    "t" := ("x" - "g1_6"["lo"]) / ("g1_6"["hi"] - "g1_6"["lo"] + 1.0E-10);
    "class_1" := "class_1" + ("t1_1_6"["lo"] * (1.0 - "t") + "t1_1_6"["hi"] * "t");
    "class_2" := "class_2" + ("t1_2_6"["lo"] * (1.0 - "t") + "t1_2_6"["hi"] * "t");
    "class_3" := "class_3" + ("t1_3_6"["lo"] * (1.0 - "t") + "t1_3_6"["hi"] * "t");
    "class_4" := "class_4" + ("t1_4_6"["lo"] * (1.0 - "t") + "t1_4_6"["hi"] * "t");
    // input 7: binary search on L1 grid
    "lo" := 0; "hi" := 15;
    "x" := "h1_7";
    IF "x" < -3.15 THEN "x" := -3.15; END_IF;
    IF "x" > 3.15 THEN "x" := 3.15; END_IF;
    WHILE "hi" - "lo" > 1 DO
        "mid" := "lo" + ("hi" - "lo") / 2;
        IF "x" > "g1_7"["mid"] THEN "lo" := "mid"; ELSE "hi" := "mid"; END_IF;
    END_WHILE;
    "t" := ("x" - "g1_7"["lo"]) / ("g1_7"["hi"] - "g1_7"["lo"] + 1.0E-10);
    "class_1" := "class_1" + ("t1_1_7"["lo"] * (1.0 - "t") + "t1_1_7"["hi"] * "t");
    "class_2" := "class_2" + ("t1_2_7"["lo"] * (1.0 - "t") + "t1_2_7"["hi"] * "t");
    "class_3" := "class_3" + ("t1_3_7"["lo"] * (1.0 - "t") + "t1_3_7"["hi"] * "t");
    "class_4" := "class_4" + ("t1_4_7"["lo"] * (1.0 - "t") + "t1_4_7"["hi"] * "t");
    // input 8: binary search on L1 grid
    "lo" := 0; "hi" := 15;
    "x" := "h1_8";
    IF "x" < -3.15 THEN "x" := -3.15; END_IF;
    IF "x" > 3.15 THEN "x" := 3.15; END_IF;
    WHILE "hi" - "lo" > 1 DO
        "mid" := "lo" + ("hi" - "lo") / 2;
        IF "x" > "g1_8"["mid"] THEN "lo" := "mid"; ELSE "hi" := "mid"; END_IF;
    END_WHILE;
    "t" := ("x" - "g1_8"["lo"]) / ("g1_8"["hi"] - "g1_8"["lo"] + 1.0E-10);
    "class_1" := "class_1" + ("t1_1_8"["lo"] * (1.0 - "t") + "t1_1_8"["hi"] * "t");
    "class_2" := "class_2" + ("t1_2_8"["lo"] * (1.0 - "t") + "t1_2_8"["hi"] * "t");
    "class_3" := "class_3" + ("t1_3_8"["lo"] * (1.0 - "t") + "t1_3_8"["hi"] * "t");
    "class_4" := "class_4" + ("t1_4_8"["lo"] * (1.0 - "t") + "t1_4_8"["hi"] * "t");
    // input 9: binary search on L1 grid
    "lo" := 0; "hi" := 15;
    "x" := "h1_9";
    IF "x" < -3.15 THEN "x" := -3.15; END_IF;
    IF "x" > 3.15 THEN "x" := 3.15; END_IF;
    WHILE "hi" - "lo" > 1 DO
        "mid" := "lo" + ("hi" - "lo") / 2;
        IF "x" > "g1_9"["mid"] THEN "lo" := "mid"; ELSE "hi" := "mid"; END_IF;
    END_WHILE;
    "t" := ("x" - "g1_9"["lo"]) / ("g1_9"["hi"] - "g1_9"["lo"] + 1.0E-10);
    "class_1" := "class_1" + ("t1_1_9"["lo"] * (1.0 - "t") + "t1_1_9"["hi"] * "t");
    "class_2" := "class_2" + ("t1_2_9"["lo"] * (1.0 - "t") + "t1_2_9"["hi"] * "t");
    "class_3" := "class_3" + ("t1_3_9"["lo"] * (1.0 - "t") + "t1_3_9"["hi"] * "t");
    "class_4" := "class_4" + ("t1_4_9"["lo"] * (1.0 - "t") + "t1_4_9"["hi"] * "t");
    // input 10: binary search on L1 grid
    "lo" := 0; "hi" := 15;
    "x" := "h1_10";
    IF "x" < -3.15 THEN "x" := -3.15; END_IF;
    IF "x" > 3.15 THEN "x" := 3.15; END_IF;
    WHILE "hi" - "lo" > 1 DO
        "mid" := "lo" + ("hi" - "lo") / 2;
        IF "x" > "g1_10"["mid"] THEN "lo" := "mid"; ELSE "hi" := "mid"; END_IF;
    END_WHILE;
    "t" := ("x" - "g1_10"["lo"]) / ("g1_10"["hi"] - "g1_10"["lo"] + 1.0E-10);
    "class_1" := "class_1" + ("t1_1_10"["lo"] * (1.0 - "t") + "t1_1_10"["hi"] * "t");
    "class_2" := "class_2" + ("t1_2_10"["lo"] * (1.0 - "t") + "t1_2_10"["hi"] * "t");
    "class_3" := "class_3" + ("t1_3_10"["lo"] * (1.0 - "t") + "t1_3_10"["hi"] * "t");
    "class_4" := "class_4" + ("t1_4_10"["lo"] * (1.0 - "t") + "t1_4_10"["hi"] * "t");
    // input 11: binary search on L1 grid
    "lo" := 0; "hi" := 15;
    "x" := "h1_11";
    IF "x" < -3.15 THEN "x" := -3.15; END_IF;
    IF "x" > 3.15 THEN "x" := 3.15; END_IF;
    WHILE "hi" - "lo" > 1 DO
        "mid" := "lo" + ("hi" - "lo") / 2;
        IF "x" > "g1_11"["mid"] THEN "lo" := "mid"; ELSE "hi" := "mid"; END_IF;
    END_WHILE;
    "t" := ("x" - "g1_11"["lo"]) / ("g1_11"["hi"] - "g1_11"["lo"] + 1.0E-10);
    "class_1" := "class_1" + ("t1_1_11"["lo"] * (1.0 - "t") + "t1_1_11"["hi"] * "t");
    "class_2" := "class_2" + ("t1_2_11"["lo"] * (1.0 - "t") + "t1_2_11"["hi"] * "t");
    "class_3" := "class_3" + ("t1_3_11"["lo"] * (1.0 - "t") + "t1_3_11"["hi"] * "t");
    "class_4" := "class_4" + ("t1_4_11"["lo"] * (1.0 - "t") + "t1_4_11"["hi"] * "t");
    // input 12: binary search on L1 grid
    "lo" := 0; "hi" := 15;
    "x" := "h1_12";
    IF "x" < -3.15 THEN "x" := -3.15; END_IF;
    IF "x" > 3.15 THEN "x" := 3.15; END_IF;
    WHILE "hi" - "lo" > 1 DO
        "mid" := "lo" + ("hi" - "lo") / 2;
        IF "x" > "g1_12"["mid"] THEN "lo" := "mid"; ELSE "hi" := "mid"; END_IF;
    END_WHILE;
    "t" := ("x" - "g1_12"["lo"]) / ("g1_12"["hi"] - "g1_12"["lo"] + 1.0E-10);
    "class_1" := "class_1" + ("t1_1_12"["lo"] * (1.0 - "t") + "t1_1_12"["hi"] * "t");
    "class_2" := "class_2" + ("t1_2_12"["lo"] * (1.0 - "t") + "t1_2_12"["hi"] * "t");
    "class_3" := "class_3" + ("t1_3_12"["lo"] * (1.0 - "t") + "t1_3_12"["hi"] * "t");
    "class_4" := "class_4" + ("t1_4_12"["lo"] * (1.0 - "t") + "t1_4_12"["hi"] * "t");
    // input 13: binary search on L1 grid
    "lo" := 0; "hi" := 15;
    "x" := "h1_13";
    IF "x" < -3.15 THEN "x" := -3.15; END_IF;
    IF "x" > 3.15 THEN "x" := 3.15; END_IF;
    WHILE "hi" - "lo" > 1 DO
        "mid" := "lo" + ("hi" - "lo") / 2;
        IF "x" > "g1_13"["mid"] THEN "lo" := "mid"; ELSE "hi" := "mid"; END_IF;
    END_WHILE;
    "t" := ("x" - "g1_13"["lo"]) / ("g1_13"["hi"] - "g1_13"["lo"] + 1.0E-10);
    "class_1" := "class_1" + ("t1_1_13"["lo"] * (1.0 - "t") + "t1_1_13"["hi"] * "t");
    "class_2" := "class_2" + ("t1_2_13"["lo"] * (1.0 - "t") + "t1_2_13"["hi"] * "t");
    "class_3" := "class_3" + ("t1_3_13"["lo"] * (1.0 - "t") + "t1_3_13"["hi"] * "t");
    "class_4" := "class_4" + ("t1_4_13"["lo"] * (1.0 - "t") + "t1_4_13"["hi"] * "t");
    // input 14: binary search on L1 grid
    "lo" := 0; "hi" := 15;
    "x" := "h1_14";
    IF "x" < -3.15 THEN "x" := -3.15; END_IF;
    IF "x" > 3.15 THEN "x" := 3.15; END_IF;
    WHILE "hi" - "lo" > 1 DO
        "mid" := "lo" + ("hi" - "lo") / 2;
        IF "x" > "g1_14"["mid"] THEN "lo" := "mid"; ELSE "hi" := "mid"; END_IF;
    END_WHILE;
    "t" := ("x" - "g1_14"["lo"]) / ("g1_14"["hi"] - "g1_14"["lo"] + 1.0E-10);
    "class_1" := "class_1" + ("t1_1_14"["lo"] * (1.0 - "t") + "t1_1_14"["hi"] * "t");
    "class_2" := "class_2" + ("t1_2_14"["lo"] * (1.0 - "t") + "t1_2_14"["hi"] * "t");
    "class_3" := "class_3" + ("t1_3_14"["lo"] * (1.0 - "t") + "t1_3_14"["hi"] * "t");
    "class_4" := "class_4" + ("t1_4_14"["lo"] * (1.0 - "t") + "t1_4_14"["hi"] * "t");
    // input 15: binary search on L1 grid
    "lo" := 0; "hi" := 15;
    "x" := "h1_15";
    IF "x" < -3.15 THEN "x" := -3.15; END_IF;
    IF "x" > 3.15 THEN "x" := 3.15; END_IF;
    WHILE "hi" - "lo" > 1 DO
        "mid" := "lo" + ("hi" - "lo") / 2;
        IF "x" > "g1_15"["mid"] THEN "lo" := "mid"; ELSE "hi" := "mid"; END_IF;
    END_WHILE;
    "t" := ("x" - "g1_15"["lo"]) / ("g1_15"["hi"] - "g1_15"["lo"] + 1.0E-10);
    "class_1" := "class_1" + ("t1_1_15"["lo"] * (1.0 - "t") + "t1_1_15"["hi"] * "t");
    "class_2" := "class_2" + ("t1_2_15"["lo"] * (1.0 - "t") + "t1_2_15"["hi"] * "t");
    "class_3" := "class_3" + ("t1_3_15"["lo"] * (1.0 - "t") + "t1_3_15"["hi"] * "t");
    "class_4" := "class_4" + ("t1_4_15"["lo"] * (1.0 - "t") + "t1_4_15"["hi"] * "t");
    // input 16: binary search on L1 grid
    "lo" := 0; "hi" := 15;
    "x" := "h1_16";
    IF "x" < -3.15 THEN "x" := -3.15; END_IF;
    IF "x" > 3.15 THEN "x" := 3.15; END_IF;
    WHILE "hi" - "lo" > 1 DO
        "mid" := "lo" + ("hi" - "lo") / 2;
        IF "x" > "g1_16"["mid"] THEN "lo" := "mid"; ELSE "hi" := "mid"; END_IF;
    END_WHILE;
    "t" := ("x" - "g1_16"["lo"]) / ("g1_16"["hi"] - "g1_16"["lo"] + 1.0E-10);
    "class_1" := "class_1" + ("t1_1_16"["lo"] * (1.0 - "t") + "t1_1_16"["hi"] * "t");
    "class_2" := "class_2" + ("t1_2_16"["lo"] * (1.0 - "t") + "t1_2_16"["hi"] * "t");
    "class_3" := "class_3" + ("t1_3_16"["lo"] * (1.0 - "t") + "t1_3_16"["hi"] * "t");
    "class_4" := "class_4" + ("t1_4_16"["lo"] * (1.0 - "t") + "t1_4_16"["hi"] * "t");

END_FUNCTION_BLOCK

// WCET estimate: L0 = 448 edges x 12 harmonics x (SIN+COS)
//   + 448 SiLU (EXP) + L1 = 64 LUT evals